TYPE (* Funk DI Struct Dual *)
  (* Version 1.0, 2026-05-28, franz *)
  PACKAGE Funk::io::DI;
  IMPORT eclipse4diac::core::TypeHash;
  IMPORT Funk::io::DI::Funk_DI_S;
  Funk_DI_S_Dual : STRUCT
    Up : Funk::io::DI::Funk_DI_S := (Pin := 127); (* forward, up, right, clockwise *)
    Down : Funk::io::DI::Funk_DI_S := (Pin := 127); (* backward, down, left, counter-clockwise *)
  END_STRUCT;
END_TYPE
